(* IEC 61131-3 sources: teller/JD_Teller_LC2_V11/Class/BoxGenerator, 1 file *)

(* ---- BoxGenerator.st ---- *)
(*!
<Class
	Name               = "BoxGenerator"
	Revision           = "1.0"
	RealtimeTask       = "true"
	CyclicTask         = "true"
	BackgroundTask     = "false"
	Sigmatek           = "false"
	OSInterface        = "false"
	HighPriority       = "false"
	Automatic          = "false"
	UpdateMode         = "Prescan"
	SharedCommandTable = "true"
	Objectsize         = "(570,540)">
	<Channels>
		<Server Name="ClassSvr" Visualized="false" Initialize="false" WriteProtected="true" Retentive="false"/>
		<Server Name="DoosLengte" Visualized="false" Initialize="false" WriteProtected="false" Retentive="false"/>
		<Server Name="GapBetweenBoxes" Visualized="false" Initialize="false" WriteProtected="false" Retentive="false"/>
		<Server Name="NrOfHoles" Visualized="false" Initialize="false" WriteProtected="false" Retentive="false"/>
		<Server Name="OneBox" Visualized="false" Initialize="false" WriteProtected="false" Retentive="false"/>
		<Server Name="OnOff" Visualized="false" Initialize="false" WriteProtected="false" Retentive="false"/>
		<Server Name="oSpeed" Visualized="true" Initialize="false" WriteProtected="true" Retentive="false"/>
		<Server Name="SensorOut" Visualized="false" Initialize="false" WriteProtected="true" Retentive="false"/>
		<Server Name="SimSpeed" Visualized="false" Initialize="false" WriteProtected="false" Retentive="false"/>
		<Server Name="TaskOnOff" Visualized="false" Initialize="false" WriteProtected="false" Retentive="false"/>
		<Client Name="c_SpeedIn" Required="false" Internal="false"/>
		<Client Name="iEncoder" Required="false" Internal="false"/>
		<Client Name="rDooslengte" Required="true" Internal="true"/>
		<Client Name="rGapBetweenBoxes" Required="true" Internal="true"/>
		<Client Name="rNrOfHoles" Required="true" Internal="true"/>
		<Client Name="rOnOff" Required="true" Internal="true"/>
	</Channels>
	<RevDoku>
		<Owner Company="JD" Author="JVD"/>
		<Dokumentation Revision="1.0" Date="2012-07-04" Author="JVD" Company="JD" Description="Taskmanager included"/>
	</RevDoku>
	<Network Name="BoxGenerator">
		<!-- List of Components in this network -->
		<Components>
			<Object
				Name       = "rDooslengte"
				Class      = "Ram"
				Position   = "(300,630)"
				Visualized = "true">
				<Channels>
					<Server Name="Data"/>
				</Channels>
			</Object>
			<Object
				Name       = "rGapBetweenBoxes"
				Class      = "Ram"
				Position   = "(300,930)"
				Visualized = "true">
				<Channels>
					<Server Name="Data"/>
				</Channels>
			</Object>
			<Object
				Name       = "rNrOfHoles"
				Class      = "Ram"
				Position   = "(300,780)"
				Visualized = "true">
				<Channels>
					<Server Name="Data"/>
				</Channels>
			</Object>
			<Object
				Name       = "rOnOff"
				Class      = "Ram"
				Position   = "(300,480)"
				Visualized = "true">
				<Channels>
					<Server Name="Data"/>
				</Channels>
			</Object>
		</Components>
		<Comments>
		</Comments>
		<!-- List of Connections in this network -->
		<Connections>
			<Connection Source="this.rOnOff" Destination="rOnOff.Data"/>
			<Connection Source="this.rDooslengte" Destination="rDooslengte.Data"/>
			<Connection Source="this.rNrOfHoles" Destination="rNrOfHoles.Data"/>
			<Connection Source="this.rGapBetweenBoxes" Destination="rGapBetweenBoxes.Data"/>
		</Connections>
		<!-- Headerfiles -->
		<Options>
		</Options>
	</Network>
</Class>
*)
BoxGenerator : CLASS
  //Servers:
	ClassSvr 	: SvrChCmd_DINT;
	TaskOnOff 	: SvrCh_DINT;
	oSpeed 	: SvrCh_DINT;
	SensorOut 	: SvrCh_DINT;
	SimSpeed 	: SvrCh_DINT;
	OnOff 	: SvrCh_DINT;
	OneBox 	: SvrCh_DINT;
	DoosLengte 	: SvrCh_DINT;
	NrOfHoles 	: SvrCh_DINT;
	GapBetweenBoxes 	: SvrCh_DINT;
  //Clients:
	iEncoder 	: CltCh_DINT;
	rOnOff 	: CltChCmd_Ram;
	rDooslengte 	: CltChCmd_Ram;
	rNrOfHoles 	: CltChCmd_Ram;
	rGapBetweenBoxes 	: CltChCmd_Ram;
	c_SpeedIn 	: CltCh_DINT;
  //Variables:
		Enc 	: Encoder1;
		BoxLength 	: DINT;
		BoxPart 	: DINT;
		BoxTeller 	: DINT;
		BoxGap 	: DINT;
		CaseOneBox 	: DINT;
		CaseBox 	: DINT;
		change 	: DINT;
  //Functions:

	FUNCTION VIRTUAL GLOBAL Init;

	FUNCTION VIRTUAL GLOBAL CyWork
		VAR_INPUT
			EAX 	: UDINT;
		END_VAR
		VAR_OUTPUT
			state (EAX) 	: UDINT;
		END_VAR;

	FUNCTION VIRTUAL GLOBAL RtWork
		VAR_INPUT
			EAX 	: UDINT;
		END_VAR
		VAR_OUTPUT
			state (EAX) 	: UDINT;
		END_VAR;

	FUNCTION VIRTUAL GLOBAL SimSpeed::Write
		VAR_INPUT
			input (EAX) 	: DINT;
		END_VAR
		VAR_OUTPUT
			result (EAX) 	: DINT;
		END_VAR;

	FUNCTION VIRTUAL GLOBAL OnOff::Write
		VAR_INPUT
			input (EAX) 	: DINT;
		END_VAR
		VAR_OUTPUT
			result (EAX) 	: DINT;
		END_VAR;

	FUNCTION VIRTUAL GLOBAL OneBox::Write
		VAR_INPUT
			input (EAX) 	: DINT;
		END_VAR
		VAR_OUTPUT
			result (EAX) 	: DINT;
		END_VAR;

	FUNCTION VIRTUAL GLOBAL DoosLengte::Write
		VAR_INPUT
			input (EAX) 	: DINT;
		END_VAR
		VAR_OUTPUT
			result (EAX) 	: DINT;
		END_VAR;

	FUNCTION VIRTUAL GLOBAL NrOfHoles::Write
		VAR_INPUT
			input (EAX) 	: DINT;
		END_VAR
		VAR_OUTPUT
			result (EAX) 	: DINT;
		END_VAR;

	FUNCTION VIRTUAL GLOBAL GapBetweenBoxes::Write
		VAR_INPUT
			input (EAX) 	: DINT;
		END_VAR
		VAR_OUTPUT
			result (EAX) 	: DINT;
		END_VAR;
  //Tables:
	FUNCTION @STD
		VAR_OUTPUT
			ret_code	: CONFSTATES;
		END_VAR;
	FUNCTION GLOBAL TAB @CT_;
END_CLASS;

#pragma using Ram

FUNCTION VIRTUAL GLOBAL BoxGenerator::Init

if    _FirstScan then

      //encoder settings
      Enc.Multi   := 1000;
      Enc.Divider := 60000*mcres;

      rOnOff  := rOnOff.Read();
      OnOff.Write(input:=rOnOff);

      rDoosLengte := rDoosLengte.Read();
      DoosLengte.Write(input:=rDoosLengte);

      rNrOfHoles := rNrOfHoles.Read();
      NrOfHoles.Write(input:=rNrOfHoles);

      rGapBetweenBoxes := rGapBetweenBoxes.Read();
      GapBetweenBoxes.Write(input:=rGapBetweenBoxes);
      BoxPart := 1;

end_if;

END_FUNCTION

FUNCTION VIRTUAL GLOBAL BoxGenerator::RtWork
	VAR_INPUT
		EAX 	: UDINT;
	END_VAR
	VAR_OUTPUT
		state (EAX) 	: UDINT;
	END_VAR

//Als in de machine setup de functie is geselelecteerd wordt de code uitgevoerd
  if  TaskOnOff then

      //Speed inlezen en omzetten naar een telwaarde
      if SimSpeed = 0 then
         c_SpeedIn := c_SpeedIn.Read();
         iEncoder += c_SpeedIn;
      else
         iEncoder += SimSpeed * MCRES;
      end_if;

      Enc.EncoderDelta := iEncoder - Enc.EncoderOld;
      Enc.EncoderOld := iEncoder;
      Enc.SpeedDelta := ((Enc.EncoderDelta * encres * enc.Multi) / enc.Divider);

      if     OneBox then

             case CaseOneBox of
             0:
                 OnOff.Write(input:=0);
                 BoxTeller := 0;
                 CaseOneBox += 1;
                 SensorOut := 0;
             1:
                 BoxTeller += Enc.SpeedDelta;
                 if ((BoxTeller/BoxPart) and 16#0001) then
                    SensorOut := 0;
                 else
                    SensorOut := 1;
                 end_if;

                 if   BoxTeller > BoxLength then
                      CaseOneBox := 2;
                      SensorOut := 0;
                 end_if;
             2:
                 OneBox := 0;
                 CaseOneBox :=0;
             end_case;
      end_if;

      if     OnOff then

             case CaseBox of
             0:
                 OneBox.Write(input:=0);
                 BoxTeller := 0;
                 CaseBox += 1;
                 SensorOut := 0;
             1:
                 BoxTeller += Enc.SpeedDelta;
                 if ((BoxTeller/BoxPart) and 16#0001) then
                    SensorOut := 0;
                 else
                    SensorOut := 1;
                 end_if;

                 if   BoxTeller > BoxLength then
                      CaseBox := 2;
                      SensorOut := 0;
                      BoxTeller := 0;
                 end_if;
             2:
                 BoxTeller += Enc.SpeedDelta;
                 if   BoxTeller > BoxGap then
                      CaseBox := 0;
                 end_if;
             end_case;
      end_if;

  end_if;

	state := READY;

END_FUNCTION

FUNCTION VIRTUAL GLOBAL BoxGenerator::CyWork
	VAR_INPUT
		EAX 	: UDINT;
	END_VAR
	VAR_OUTPUT
		state (EAX) 	: UDINT;
	END_VAR

//Als in de machine setup de functie is geselelecteerd wordt de code uitgevoerd
  if  TaskOnOff then

      //Snelheidsberekening
      oSpeed := c_SpeedIn/mcres;

      if change then
        if  NrOfHoles > 0 then
          BoxPart := (DoosLengte*encres) / ((NrOfHoles * 2) + 1);
          BoxLength := DoosLengte*encres;
          BoxGap := GapBetweenBoxes * encres;
        else
          BoxLength := DoosLengte*encres;
          BoxPart := BoxLength;
          BoxGap := GapBetweenBoxes * encres;
        end_if;
        change :=0;
      end_if;

  end_if;
	state := READY;

END_FUNCTION

FUNCTION VIRTUAL GLOBAL BoxGenerator::OnOff::Write
	VAR_INPUT
		input (EAX) 	: DINT;
	END_VAR
	VAR_OUTPUT
		result (EAX) 	: DINT;
	END_VAR

	OnOff := input;
  if  OnOff < 0 | OnOff > 1 then
      OnOff := 0;
  end_if;
  SensorOut := 0;
  rOnOff.Write(input:=OnOff);

 	result := OnOff;

END_FUNCTION

FUNCTION VIRTUAL GLOBAL BoxGenerator::OneBox::Write
	VAR_INPUT
		input (EAX) 	: DINT;
	END_VAR
	VAR_OUTPUT
		result (EAX) 	: DINT;
	END_VAR

	OneBox := input;
  if OneBox < 0 | OneBox > 1 then
     OneBox := 0;
  end_if;
  SensorOut := 0;
 	result := OneBox;

END_FUNCTION

FUNCTION VIRTUAL GLOBAL BoxGenerator::DoosLengte::Write
	VAR_INPUT
		input (EAX) 	: DINT;
	END_VAR
	VAR_OUTPUT
		result (EAX) 	: DINT;
	END_VAR

	DoosLengte := input;
  if DoosLengte < 100 then
     DoosLengte := 100;
  elsif DoosLengte > 2000 then
        DoosLengte := 2000;
  end_if;

  rDooslengte.Write(input:=DoosLengte);
  change := 1;

 	result := DoosLengte;

END_FUNCTION

FUNCTION VIRTUAL GLOBAL BoxGenerator::NrOfHoles::Write
	VAR_INPUT
		input (EAX) 	: DINT;
	END_VAR
	VAR_OUTPUT
		result (EAX) 	: DINT;
	END_VAR

	NrOfHoles := input;
  if NrOfHoles < 0 then
     NrOfHoles := 0;
  elsif NrOfHoles > 8 then
        NrOfHoles := 8;
  end_if;

  rNrOfHoles.Write(input:=NrOfHoles);
  change := 1;

 	result := NrOfHoles;

END_FUNCTION

FUNCTION VIRTUAL GLOBAL BoxGenerator::GapBetweenBoxes::Write
	VAR_INPUT
		input (EAX) 	: DINT;
	END_VAR
	VAR_OUTPUT
		result (EAX) 	: DINT;
	END_VAR

	GapBetweenBoxes := input;
  if    GapBetweenBoxes < 50 then
        GapBetweenBoxes := 50;
  elsif GapBetweenBoxes > 2000 then
        GapBetweenBoxes := 2000;
  end_if;

  rGapBetweenBoxes.Write(input:=GapBetweenBoxes);
  change := 1;
 	result := GapBetweenBoxes;

END_FUNCTION

FUNCTION VIRTUAL GLOBAL BoxGenerator::SimSpeed::Write
	VAR_INPUT
		input (EAX) 	: DINT;
	END_VAR
	VAR_OUTPUT
		result (EAX) 	: DINT;
	END_VAR

	SimSpeed := input;
  if  SimSpeed < 0 then
      SimSpeed := 0;
  end_if;

 	result := SimSpeed;

END_FUNCTION
